Universal Robots URScript: 00C_01_ZhuaXian.script

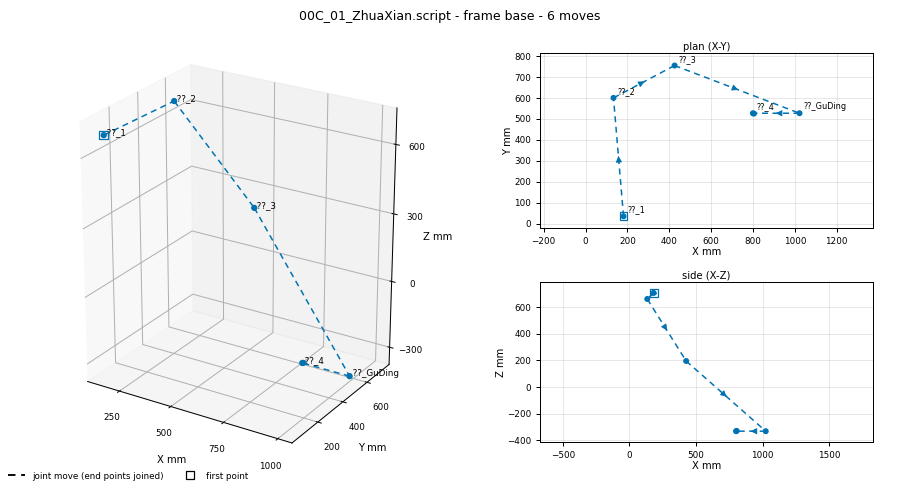
[picture p0: tool path of 00C_01_ZhuaXian.script in frame base, 6 of 6 moves have a stored position in this frame; points joined in program order, loops and branches not executed]
def P00C_01_ZhuaXian():
  set_standard_analog_input_domain(0, 1)
  set_standard_analog_input_domain(1, 1)
  set_tool_analog_input_domain(0, 1)
  set_tool_analog_input_domain(1, 1)
  set_analog_outputdomain(0, 0)
  set_analog_outputdomain(1, 0)
  set_tool_voltage(0)
  set_input_actions_to_default()
  set_tcp(p[-0.06448999999999999,0.0207,0.28314999999999996,0.0,0.0,1.5902])
  set_payload(8.0)
  set_safety_mode_transition_hardness(1)
  set_gravity([0.0, 0.0, 9.82])
  $ 1 "机器人程序"
  $ 2 "MoveJ"
  $ 3 "路点_1"
  set_tcp(p[-8.5E-4,0.01448,0.31003,0.0,0.0,-0.3645])
  movej(get_inverse_kin(p[.181493968573, .034606211380, .705741013575, .017056972338, .054038250851, -1.587611529093], qnear=[1.6280300617218018, 0.05505633354187012, -2.8315115610705774, -1.8881071249591272, -1.5483978430377405, -4.423880640660421]), a=0.6981317007977318, v=0.5235987755982988)
  $ 4 "路点_2"
  set_tcp(p[-8.5E-4,0.01448,0.31003,0.0,0.0,-0.3645])
  movej(get_inverse_kin(p[.133452865962, .600641103194, .660554241773, -.045945149075, .048976497060, .006624512094], qnear=[1.640486478805542, -1.7533162275897425, -2.3389506975757044, -0.6614764372455042, -1.5246756712542933, -2.840433184300558]), a=0.6981317007977318, v=0.5235987755982988)
  $ 5 "路点_3"
  set_tcp(p[-8.5E-4,0.01448,0.31003,0.0,0.0,-0.3645])
  movej(get_inverse_kin(p[.425276578395, .755226957564, .195084053182, -.266065499907, 1.522738494105, .032011131546], qnear=[1.761915922164917, -1.9969714323626917, -2.209606472645895, -0.5377591292010706, -0.03227550188173467, -2.898017708455221]), a=0.6981317007977318, v=0.5235987755982988)
  $ 6 "路点_GuDing"
  set_tcp(p[-8.5E-4,0.01448,0.31003,0.0,0.0,-0.3645])
  movej(get_inverse_kin(p[1.022356227480, .527263301860, -.331224856978, .093642636484, 1.562847395811, -.207671855129], qnear=[0.9411043524742126, -2.871925179158346, -1.3866542021380823, -1.9792006651507776, -0.4444053808795374, -1.3238518873797815]), a=0.6981317007977318, v=0.5235987755982988)
  $ 7 "路点_4"
  set_tcp(p[-8.5E-4,0.01448,0.31003,0.0,0.0,-0.3645])
  movej(get_inverse_kin(p[.799563753343, .527188886284, -.331300849798, .093688867516, 1.562902298711, -.207758744609], qnear=[1.195081114768982, -2.792774025593893, -1.7243498007403772, -1.6699779669391077, -0.19034940401186162, -1.3743374983416956]), a=0.6981317007977318, v=0.5235987755982988)
  $ 8 "路点_5"
  set_tcp(p[-8.5E-4,0.01448,0.31003,0.0,0.0,-0.3645])
  movej(get_inverse_kin(p[.804535913287, .525390225580, -.328925464284, .111200223326, 1.481237752095, -.235922417218], qnear=[1.18886137008667, -2.8590362707721155, -1.7424452940570276, -1.1460345427142542, -0.19415122667421514, -1.8057783285724085]), a=0.6981317007977318, v=0.5235987755982988)
end
